FUNCTION_BLOCK FB_AutoSwitch EXTENDS FB_BaseDevice
VAR
	bRawInput AT %I*: BOOL;
END_VAR

IF bRawInput THEN
	eState := E_DeviceState.ON;
ELSE
	eState := E_DeviceState.OFF;
END_IF

END_FUNCTION_BLOCK

(* stored: Version 1.1.0.1, ProductVersion 3.1.4024.12
   POU FB_AutoSwitch: Id {397fde9c-1482-401d-b372-27dcab041960}, SpecialFunc None *)
